Staubli VAL3: JointTrajPtMsg.pjx

--- JointTrajPtMsg.pjx ---
Parameters version=s7.7.2 stackSize=5000 millimeterUnit=true
Program file=start.pgx
Program file=stop.pgx
Data file=JointTrajPtMsg.dtx
Type name=Body path=Disk://ros_libs/Body/Body.pjx
Type name=Header path=Disk://ros_libs/Header/Header.pjx
Type name=Prefix path=Disk://ros_libs/Prefix/Prefix.pjx
Type name=JointTrajPt path=Disk://ros_libs/JointTrajPt/JointTrajPt.pjx

--- JointTrajPtMsg.dtx ---
public Header header
  [0]
    num nMsgType
    num nCommType
    num nReplyCode
    num nData[12]
public JointTrajPt jointTrajPt
  [0]
    num nSeq
    num nJoints[10]
    num nVelocity
    num nDuration
public Prefix prefix
  [0]
    num nLength
    num nData[4]
public Body body
  [0]
    num nData[64]
